// TwinCAT 3 PLC project PLC1
// ProgramVersion: 3.1.4024.0
// libraries:
//   Tc2_Standard, * (Beckhoff Automation GmbH)
//   Tc2_System, * (Beckhoff Automation GmbH)
//   Tc3_Module, * (Beckhoff Automation GmbH)
// project tree:
//   GVLs/ GVL_ADS.TcGVL, GVL_IO.TcGVL
//   / PlcTask.TcTTO (not stored)
//   POUs/ MAIN.TcPOU
// real-time tasks:
//   TASK PlcTask: cycle T#10ms, priority 20, ADS port 350
// I/O:
//   DEVICE Device 1 (CX-BK)
//     Box 1 (CX-BK)
//   DEVICE Device 2 (NOV-DP-RAM)
//   DEVICE Device 3 (CX7000), AmsNetId 5.129.88.118.4.1
//     Term 3 (CX7028) [CX7028-0000-0118]
//       modules: Module 1 (DIO_2x), Module 3 (DIO_2x), Module 5 (DI_2x), Module 7 (DI_2x)
// variable links:
//   PLC1/PLC1 Instance <-> Device 1 (CX-BK)/Box 1 (CX-BK)
//     PlcTask Inputs/GVL_IO.iInput <-> Term 2 (KL3062)/Channel 1/Data In

// ---- GVLs/GVL_ADS.TcGVL
{attribute 'Tc2GvlVarNames'}
VAR_GLOBAL
	Array_EPB_TDA_INT AT%MB1100	: ARRAY [0..20] OF INT;
	ArrayReceiveWrite 			: ARRAY [0..20] OF INT;
END_VAR

// ---- GVLs/GVL_IO.TcGVL
{attribute 'qualified_only'}
VAR_GLOBAL
	iInput AT%I* : INT;
END_VAR

// ---- POUs/MAIN.TcPOU
PROGRAM MAIN
VAR
	i: INT;
	// Variable to Cycle ADS Values
	bEven: BOOL := 0;
END_VAR

IF bEven THEN		
	FOR i := 0 TO 20 DO
		GVL_ADS.Array_EPB_TDA_INT[i] := i*20;
		bEven := FALSE;
	END_FOR
ELSE
	FOR i := 0 TO 20 DO
		GVL_ADS.Array_EPB_TDA_INT[i] := i*10;
		bEven := TRUE;
	END_FOR
END_IF

END_PROGRAM
